(* IEC 61131-3 sources: inproshop/Team-Test20_exported/OP70/2.PRG, 8 files *)

(* ---- OP70_Communication.st ---- *)
PROGRAM OP70_Communication
VAR
	OP08HeartdelayON:TON;
	OP08HeartdelayOFF:TON;
	MasterHeartdelayON:TON;
	MasterHeartdelayOFF:TON;
END_VAR

//心跳输出
IF CPU_Clock.Clock_1s THEN
	DB7005_Communication.TO_OPXX.Heart:=1;
ELSE
	DB7005_Communication.TO_OPXX.Heart:=0;
END_IF

OP08HeartdelayON(IN:= DB7005_Communication.From_OPXX.Heart=1, PT:= T#2S, Q=> , ET=> );
OP08HeartdelayOFF(IN:= DB7005_Communication.From_OPXX.Heart=0, PT:= T#2S, Q=> , ET=> );

//前站掉线报警
IF (OP08HeartdelayON.Q OR OP08HeartdelayOFF.Q) AND NOT DB7000_Control.Mode.Status.OfflineMode  THEN
	DB7070_Fault.Stop.BeforStation_Communication_Rrror:=TRUE;
END_IF

//主站心跳通讯检测
MasterHeartdelayON(IN:= DB7005_Communication.FromMaster.Heart=1, PT:= T#2S, Q=> , ET=> );
MasterHeartdelayOFF(IN:= DB7005_Communication.FromMaster.Heart=0, PT:= T#2S, Q=> , ET=> );
//主站掉线报警
IF (MasterHeartdelayON.Q OR MasterHeartdelayOFF.Q) AND NOT DB7000_Control.Mode.Status.OfflineMode  THEN
	DB7070_Fault.Stop.MasterTimeOut:=TRUE;
END_IF

//与主站配方不一致报警
IF DB7005_Communication.FromMaster.MasterRecipeID<>DB7002_Recipe.RecipeNum AND NOT DB7000_Control.Mode.Status.OfflineMode THEN
	DB7070_Fault.Stop.MaterReipeDiscrepancy:=TRUE;
END_IF

(* ---- OP70_Control.st ---- *)
PROGRAM OP70_Control
VAR
	FB_ModeControl_instance:FB_ModeControl_V1;
	FB_Count_instance:ARRAY[0..2] OF FB_Count;
END_VAR

(**********模式切换功能***********)
FB_ModeControl_instance(
	iClock:= CPU_Clock,
	iStartDelay:= T#0.1S,
	iEstop:=DB7070_Fault.EstopTotal,
	iAlam:=DB7070_Fault.StopTotal,
	iWarn:=DB7070_Fault.RunTotal,
	ioMachine:= DB7000_Control.Machine,
	ioMode:=DB7000_Control.Mode);

(********************计数****************************)
//总计数
FB_Count_instance[0](
	ioCount:= DB7003_Count.Total,
	iClock:= CPU_Clock,
	iDayStartTime:= CPU_Clock.DayStartTime,
	iNightStartTime:=CPU_Clock.NightStartTime);

//OK计数
FB_Count_instance[1](
	ioCount:= DB7003_Count.OK,
	iClock:= CPU_Clock,
	iDayStartTime:= CPU_Clock.DayStartTime,
	iNightStartTime:=CPU_Clock.NightStartTime);

//NG计数
FB_Count_instance[2](
	ioCount:= DB7003_Count.NG,
	iClock:= CPU_Clock,
	iDayStartTime:= CPU_Clock.DayStartTime,
	iNightStartTime:=CPU_Clock.NightStartTime);

(***********良率计算***********)
//良率统计
IF DB7003_Count.Total.Today.Total<>0 THEN
	DB7003_Count.Yield:=DB7003_Count.OK.Today.Total/DB7003_Count.Total.Today.Total;
ELSE
	DB7003_Count.Yield:=0;
END_IF
//良率清零
IF DB7003_Count.Clear THEN
	DB7003_Count.Total.Today.Total:=0;
	DB7003_Count.OK.Today.Total:=0;
	DB7003_Count.NG.Today.Total:=0;
	DB7003_Count.Clear:=FALSE;
END_IF

(********程序调用*******)
OP70_DI_Mirror();
OP70_Communication();
OP70_Recipe();
OP70_Graph();
OP70_DriveControl();
OP70_DO_Mirror();
OP70_Fault();

(* ---- OP70_DI_Mirror.st ---- *)
PROGRAM OP70_DI_Mirror
VAR
	i:INT;//循环用变量
	Page:INT;
	Monitor:ARRAY[0..15] OF Str_IOMonitor;
	Status:WORD;
	Map:BOOL;
END_VAR

ACT_MAP();
ACT_Comment();
ACT_Status();

(* ---- OP70_DO_Mirror.st ---- *)
PROGRAM OP70_DO_Mirror
VAR
	i:INT;//循环用变量
	Page:INT;
	Monitor:ARRAY[0..15] OF Str_IOMonitor;
	Status:WORD;
	Map:BOOL;
	Startlamp1:BOOL;
	Startlamp2:BOOL;
END_VAR

ACT_MAP();
ACT_Comment();
ACT_Status();

(* ---- OP70_DriveControl.st ---- *)
PROGRAM OP70_DriveControl
VAR
	FB_Cylinder_instance :ARRAY[0..63]OF FB_Cylinder_V1;
	FB_Vacuum_instance :ARRAY[0..31]OF FB_Vacuum_V1;
	FB_Axis_Instance:ARRAY[0..31]OF FB_Axis_V1_3;
	FB_Sensor_instance :ARRAY[0..63]OF FB_Sensor_V1_1;
	FB_TcpClient_Instance:ARRAY[0..31]OF FB_TcpClient;
	FB_DoubleStart_Instance:ARRAY[1..1]OF FB_DoubleStart;
	FB_Epson_V1_Instance:ARRAY[1..1]OF FB_Epson_V1;
	FB_Kuka_V1_Instance:ARRAY[1..10]OF FB_Kuka_V1;
	FB_Rotdisk_V1_Instance:ARRAY[1..1]OF FB_Rotdisk_V1;
	FB_Stopper_V1_Instance:ARRAY[1..10]OF FB_Stopper_V1;
	FB_AI_Instance:ARRAY[1..1]OF FB_AI;
	FB_Motor_Instance:ARRAY[1..1]OF FB_Motor;
	FB_Heating_Instance:ARRAY[1..1]OF FB_Heating;
	FB_Cam_Instance:ARRAY[1..1]OF FB_Cam;
	FB_AAS_Instance:ARRAY[1..1]OF FB_AAS;
	FB_ElectricScrewdriver_Instance:ARRAY[1..4]OF FB_ElectricScrewdriver_V1_1_0;
	FB_ScrewFeeder_Instance:ARRAY[1..4]OF FB_ScrewFeeder;
	FB_Code_Instance:ARRAY[1..4]OF FB_Code;
	FB_Print_Instance:ARRAY[1..1]OF FB_Print;
END_VAR
VAR
	i:INT;//循环变量用
	EpsonTcpClient:ARRAY[1..1]OF Str_TcpClient;
	KukaTcpClient:ARRAY[1..1]OF Str_TcpClient;
END_VAR

ACT_Axis();
ACT_Cylinder();
ACT_Vacuum();
ACT_Sensor();
ACT_Cam();
ACT_ElectricScrewdriver();
ACT_CODE();
ACT_Print();

(* ---- OP70_Fault.st ---- *)
PROGRAM OP70_Fault
VAR
	i:UINT;//循环变量用
	Pobool_IN: POINTER TO BOOL;//输入报警指针地址获取；
	Pobool_OUT: POINTER TO BOOL;//输出报警指针地址获取；
	EstopMAP:ARRAY[0..255] OF BOOL;
	StopMAP:ARRAY[0..999] OF BOOL;
	RunMAP:ARRAY[0..255] OF BOOL;
	Size:UINT;//数组数量
	Estop_R:R_TRIG;//急停上升沿
	Stop_R:R_TRIG;//暂停上升沿
	Run_R:R_TRIG;//警告上升沿
END_VAR

//气缸报警地址映射
SizeOfAry(In:=DB7050_DriveControl.CylCtrl,Out=>Size);
FOR i:=0 TO Size-1 BY 1 DO
	DB7070_Fault.Stop.Cyl[I]:=DB7050_DriveControl.CylCtrl[i].Status.Error;
END_FOR
//真空报警映射
SizeOfAry(In:=DB7050_DriveControl.VacCtrl,Out=>Size);
FOR i:=0 TO Size-1 BY 1 DO
	DB7070_Fault.Stop.Vac[I]:=DB7050_DriveControl.VacCtrl[i].Status.Error;
END_FOR
//轴报警映射
SizeOfAry(In:=DB7050_DriveControl.AxisCtrl,Out=>Size);
FOR i:=0 TO Size-1 BY 1 DO
	DB7070_Fault.Stop.Axis[I]:=DB7050_DriveControl.AxisCtrl[i].Status.Error;
END_FOR

//急停报警
DB7070_Fault.Estop.EstopButton:=NOT DB7000_Control.Machine.EmgSafetyRelay;

//暂停报警

//提示

ACT_MAP();
ACT_HMI_Jump();

(* ---- OP70_Graph.st ---- *)
PROGRAM OP70_Graph
VAR
	IntitalTimeDelay:ARRAY[1..9,0..10] OF TON;//初始化流程用
	AutoTimeDelay:ARRAY[1..9,0..10] OF TON;//自动流程用
	Init:ARRAY[1..20]OF Str_Graph := [20((Complete := TRUE))];//初始化
	Auto:ARRAY[1..20]OF Str_Graph;//自动
	Start:ARRAY[1..9] OF BOOL;//自动启动条件
	i:INT;//循环变量用
	Screw:ARRAY[1..4] OF Str_OP70_Screw;
END_VAR

ACT_InitST1();
ACT_InitST2();
ACT_InitST3();
ACT_InitST4();
ACT_InitST5();
ACT_InitST6();
ACT_AutoRunST1_人工上料打码();
ACT_AutoRunST2_同步搬运();
ACT_AutoRunST3_侧面1锁螺丝工位();
ACT_AutoRunST4_侧面2锁螺丝工位();
ACT_AutoRunST5_顶面锁螺丝工位();
ACT_AutoRunST6_下料工位();

(* ---- OP70_Recipe.st ---- *)
PROGRAM OP70_Recipe
VAR
	i:INT;
	DownLoad_R:R_TRIG;
	Download_F:F_TRIG;
	Change:R_TRIG;
END_VAR
VAR RETAIN PERSISTENT
	RecipeNum AT %MB131080 : INT;
END_VAR

//配方名
DB7002_Recipe.RecipeName:=DB7002_Recipe.TypeData[DB7002_Recipe.RecipeNum].Name;

//主线一键切换
IF DB7005_Communication.FromMaster.OnLineMode=1 THEN
	DB7002_Recipe.RecipeNumTemp:=DB7005_Communication.FromMaster.RecipeID;
END_IF

//配方参数修改使能
IF DB7002_Recipe.RecipeNum=DB7002_Recipe.RecipeNumTemp THEN
	DB7002_Recipe.ParameterChangePmt:=TRUE;
ELSE
	DB7002_Recipe.ParameterChangePmt:=FALSE;
END_IF

//配方允许切换使能
DB7002_Recipe.RecipeChangePmt:=DB7000_Control.Mode.Status.ManualMode OR DB7005_Communication.FromMaster.OnLineMode=1;

//配方名称获取
IF RecipeNum<>DB7002_Recipe.RecipeNumTemp THEN
	DB7002_Recipe.RecipeNameTemp:=DB7002_Recipe.TypeData[DB7002_Recipe.RecipeNumTemp].Name;
	RecipeNum:=DB7002_Recipe.RecipeNumTemp;
END_IF

DownLoad_R(CLK:= DB7002_Recipe.DownLoad OR (DB7005_Communication.FromMaster.OnLineMode=1 AND DB7005_Communication.FromMaster.RecipeDownLoad=1));
DownLoad_F(CLK:= DB7002_Recipe.DownLoad OR (DB7005_Communication.FromMaster.OnLineMode=1 AND DB7005_Communication.FromMaster.RecipeDownLoad=1));
ACT_Upload();
ACT_Download();

//一键切换配方时，从站退出初始化完成状态
IF DB7005_Communication.FromMaster.OnLineMode=1 AND DB7005_Communication.FromMaster.RecipeDownLoad=1 THEN
	DB7000_Control.Mode.Status.HomeOK:=FALSE;
	DB7000_Control.Mode.Status.AutoRunning:=FALSE;
END_IF
